// TIA Portal project "PROGETTO_TISC_FOSCHILLO_CUOMO" (V17)
// Vorlageprojekt für das Buch mit Zielsystem S7-1200

(* hardware
DEVICE "S7-1200-Station_1"  S7-1200 Station
   slot 0: "Baugruppenträger_0"  Rack  V1.0
   slot 1: "PLC_1"  CPU 1214C DC/DC/DC  6ES7 214-1AG40-0XB0  V4.5
DEVICE "HMI_1"  TP900 Comfort
   slot 0: "HMI_1"  TP900 Comfort  6AV2 124-0JC01-0AX0  17.0.0.0
   slot 1: "HMI_RT_1"  TP900 Comfort  6AV2 124-0JC01-0AX0  17.0.0.0
   slot 5: "HMI_1.IE_CP_1"  PROFINET Interface  17.0.0.0
      slot 1: "PROFINET Interface_1"  PROFINET Interface
         slot 1: "Port_1"  Port
         slot 2: "Port_2"  Port
   slot 7: "HMI_1.MPI/DP_CP_1"  MPI/DP Interface  17.0.0.0
*)

// ===== PLC "PLC_1"  CPU 1214C DC/DC/DC =====

VAR_GLOBAL   // PLC tag table "Standard-Variablentabelle"
   "Tag_1" AT %A0.0 : Bool;
   "Tag_2" AT %E0.0 : Bool;
   "Tag_3" AT %E0.1 : Bool;
   "PIANO_0" AT %I0.2 : Bool;
   "PIANO1_SLOW" AT %I0.3 : Bool;
   "PIANO1_STOP" AT %I0.4 : Bool;
   "PIANO2_SLOW" AT %I0.5 : Bool;
   "PIANO2_STOP" AT %I0.6 : Bool;
   "BASE_UP" AT %Q0.1 : Bool;
   "BASE_DOWN" AT %Q0.2 : Bool;
   "BASE_SLOW" AT %Q0.3 : Bool;
   "SENS_DX" AT %I0.7 : Bool;
   "SENS_SX" AT %I1.0 : Bool;
   "SPOSTA_DX" AT %Q0.4 : Bool;
   "SPOSTA_SX" AT %Q0.5 : Bool;
   "SPINGI_INIZIO" AT %I1.1 : Bool;
   "SPINGI_FINE" AT %I1.2 : Bool;
   "SENS_SPINGI" AT %I1.3 : Bool;
   "SPINGI" AT %Q0.6 : Bool;
   "PRONTO_CONS" AT %I1.4 : Bool;
   "AVA" AT %Q0.7 : Bool;
   "H1" AT %I1.5 : Bool;
   "H2" AT %I1.6 : Bool;
   "AVA1" AT %Q1.0 : Bool;
   "CONS_ELEV" AT %I1.7 : Bool;
   "RICEVUTO_P1" AT %I2.0 : Bool;
   "RICEVUTO_P2" AT %I2.1 : Bool;
   "AVA2" AT %Q1.1 : Bool;
   "AVA3" AT %Q1.2 : Bool;
   "Tag_4" AT %M1.0 : Bool;
   "Tag_5" AT %M1.1 : Bool;
   "pezzi_lavorati_NP1" AT %MW16 : Int;
   "pezzi_lavorati_NP2" AT %MW18 : Int;
END_VAR

DATA_BLOCK "MS0_DB"   // DB1
{ S7_Optimized_Access := 'TRUE' }
VERSION : 0.1
// stored: InstanceOfName MECCANISMO DI SPOSTAMENTO
"MECCANISMO DI SPOSTAMENTO"
BEGIN
END_DATA_BLOCK

DATA_BLOCK "P_DB"   // DB2
{ S7_Optimized_Access := 'TRUE' }
VERSION : 0.1
// stored: InstanceOfName Pusher
"Pusher"
BEGIN
END_DATA_BLOCK

DATA_BLOCK "BR0_DB"   // DB3
{ S7_Optimized_Access := 'TRUE' }
VERSION : 0.1
// stored: InstanceOfName Base con rulliera
"Base con rulliera"
BEGIN
END_DATA_BLOCK

DATA_BLOCK "N2_DB"   // DB4
{ S7_Optimized_Access := 'TRUE' }
VERSION : 0.1
// stored: InstanceOfName Nastro_2
"Nastro_2"
BEGIN
END_DATA_BLOCK

DATA_BLOCK "N1_DB"   // DB5
{ S7_Optimized_Access := 'TRUE' }
VERSION : 0.1
// stored: InstanceOfName Nastro_1
"Nastro_1"
BEGIN
END_DATA_BLOCK

DATA_BLOCK "NP1_DB"   // DB7
{ S7_Optimized_Access := 'TRUE' }
VERSION : 0.1
// stored: InstanceOfName nastri_sup
"nastri_sup"
BEGIN
END_DATA_BLOCK

DATA_BLOCK "NP2_DB"   // DB8
{ S7_Optimized_Access := 'TRUE' }
VERSION : 0.1
// stored: InstanceOfName nastri_sup
"nastri_sup"
BEGIN
END_DATA_BLOCK

DATA_BLOCK "nastri_sup_DB"   // DB9
{ S7_Optimized_Access := 'TRUE' }
VERSION : 0.1
// stored: InstanceOfName nastri_sup
"nastri_sup"
BEGIN
END_DATA_BLOCK

FUNCTION_BLOCK "MECCANISMO DI SPOSTAMENTO"   // FB1, LAD
{ S7_Optimized_Access := 'TRUE' }
VERSION : 0.1
   VAR_INPUT
      consegnato : Bool;
      ferma2 : Bool;
      ferma1 : Bool;
      PIANO_0 : Bool;
      PIANO1_SLOW : Bool;
      PIANO1_STOP : Bool;
      PIANO2_SLOW : Bool;
      sali_ok : Bool;
      PIANO2_STOP : Bool;
   END_VAR
   VAR_OUTPUT
      down_ok : Bool;
      BASE_UP : Bool;
      BASE_DOWN : Bool;
      pronto_ferma : Bool;
      BASE_SLOW : Bool;
   END_VAR
   VAR
      initVar : Bool;
      f0 : Bool;
      f1 : Bool;
      f2 : Bool;
      f3 : Bool;
      f4 : Bool;
      f5 : Bool;
      f6 : Bool;
      f7 : Bool;
      t1 : Bool;
      t2 : Bool;
      t3 : Bool;
      t4 : Bool;
      t5 : Bool;
      t6 : Bool;
      t7 : Bool;
      t8 : Bool;
      t9 : Bool;
   END_VAR
BEGIN

REGION Network 1: inizializzazione fase F0
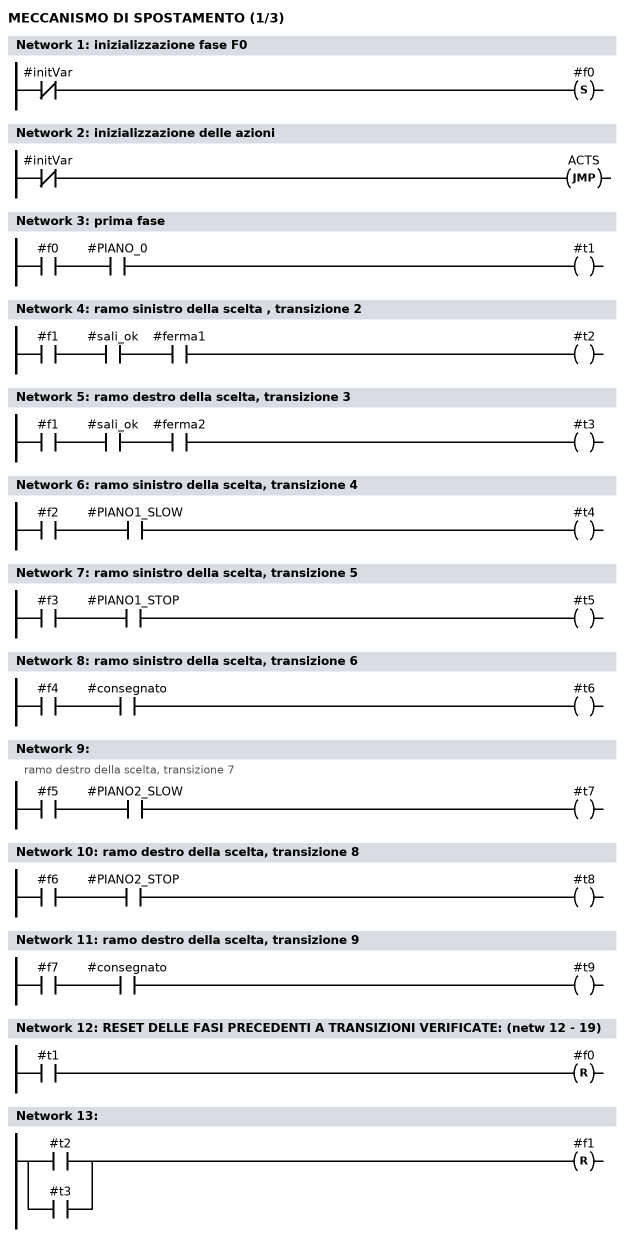
   RUNG wire#powerrail
      I_Contact( #initVar )
      S_Coil( #f0 )
   END_RUNG
   // the same network as SCL:
   IF NOT #initVar THEN #f0 := TRUE; END_IF;
END_REGION

REGION Network 2: inizializzazione delle azioni
   RUNG wire#powerrail
      I_Contact( #initVar )
      JumpCoil( ACTS )
   END_RUNG
   // the same network as SCL:
   IF NOT #initVar THEN GOTO ACTS; END_IF;
END_REGION

REGION Network 3: prima fase
   RUNG wire#powerrail
      Contact( #f0 )
      Contact( #PIANO_0 )
      Coil( #t1 )
   END_RUNG
   // the same network as SCL:
   #t1 := #f0 AND #PIANO_0;
END_REGION

REGION Network 4: ramo sinistro della scelta , transizione 2
   RUNG wire#powerrail
      Contact( #f1 )
      Contact( #sali_ok )
      Contact( #ferma1 )
      Coil( #t2 )
   END_RUNG
   // the same network as SCL:
   #t2 := #f1 AND #sali_ok AND #ferma1;
END_REGION

REGION Network 5: ramo destro della scelta, transizione 3
   RUNG wire#powerrail
      Contact( #f1 )
      Contact( #sali_ok )
      Contact( #ferma2 )
      Coil( #t3 )
   END_RUNG
   // the same network as SCL:
   #t3 := #f1 AND #sali_ok AND #ferma2;
END_REGION

REGION Network 6: ramo sinistro della scelta, transizione 4
   RUNG wire#powerrail
      Contact( #f2 )
      Contact( #PIANO1_SLOW )
      Coil( #t4 )
   END_RUNG
   // the same network as SCL:
   #t4 := #f2 AND #PIANO1_SLOW;
END_REGION

REGION Network 7: ramo sinistro della scelta, transizione 5
   RUNG wire#powerrail
      Contact( #f3 )
      Contact( #PIANO1_STOP )
      Coil( #t5 )
   END_RUNG
   // the same network as SCL:
   #t5 := #f3 AND #PIANO1_STOP;
END_REGION

REGION Network 8: ramo sinistro della scelta, transizione 6
   RUNG wire#powerrail
      Contact( #f4 )
      Contact( #consegnato )
      Coil( #t6 )
   END_RUNG
   // the same network as SCL:
   #t6 := #f4 AND #consegnato;
END_REGION

REGION Network 9
   // ramo destro della scelta, transizione 7
   RUNG wire#powerrail
      Contact( #f5 )
      Contact( #PIANO2_SLOW )
      Coil( #t7 )
   END_RUNG
   // the same network as SCL:
   #t7 := #f5 AND #PIANO2_SLOW;
END_REGION

REGION Network 10: ramo destro della scelta, transizione 8
   RUNG wire#powerrail
      Contact( #f6 )
      Contact( #PIANO2_STOP )
      Coil( #t8 )
   END_RUNG
   // the same network as SCL:
   #t8 := #f6 AND #PIANO2_STOP;
END_REGION

REGION Network 11: ramo destro della scelta, transizione 9
   RUNG wire#powerrail
      Contact( #f7 )
      Contact( #consegnato )
      Coil( #t9 )
   END_RUNG
   // the same network as SCL:
   #t9 := #f7 AND #consegnato;
END_REGION

REGION Network 12: RESET DELLE FASI PRECEDENTI A TRANSIZIONI VERIFICATE: (netw 12 - 19)
   RUNG wire#powerrail
      Contact( #t1 )
      R_Coil( #f0 )
   END_RUNG
   // the same network as SCL:
   IF #t1 THEN #f0 := FALSE; END_IF;
END_REGION

REGION Network 13
   RUNG wire#powerrail
      Contact( #t2 )
      wire#w1
      R_Coil( #f1 )
   END_RUNG
   RUNG wire#powerrail
      Contact( #t3 )
   END_RUNG wire#w1
   // the same network as SCL:
   IF #t2 OR #t3 THEN #f1 := FALSE; END_IF;
END_REGION

REGION Network 14
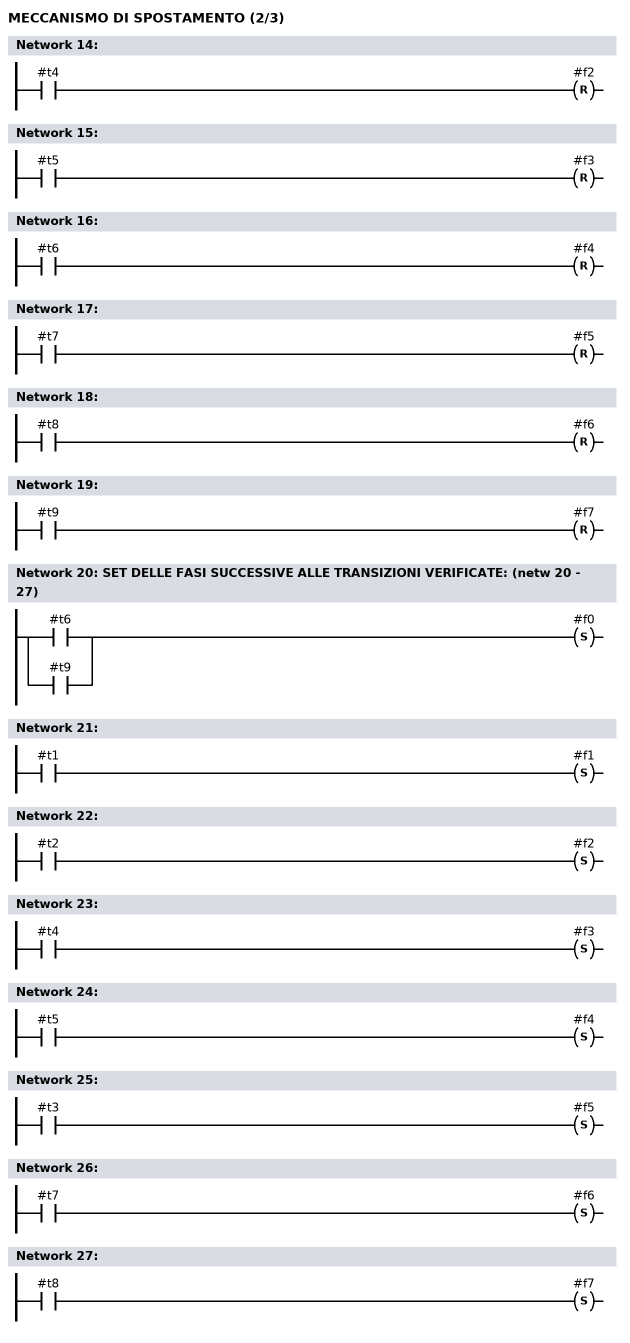
   RUNG wire#powerrail
      Contact( #t4 )
      R_Coil( #f2 )
   END_RUNG
   // the same network as SCL:
   IF #t4 THEN #f2 := FALSE; END_IF;
END_REGION

REGION Network 15
   RUNG wire#powerrail
      Contact( #t5 )
      R_Coil( #f3 )
   END_RUNG
   // the same network as SCL:
   IF #t5 THEN #f3 := FALSE; END_IF;
END_REGION

REGION Network 16
   RUNG wire#powerrail
      Contact( #t6 )
      R_Coil( #f4 )
   END_RUNG
   // the same network as SCL:
   IF #t6 THEN #f4 := FALSE; END_IF;
END_REGION

REGION Network 17
   RUNG wire#powerrail
      Contact( #t7 )
      R_Coil( #f5 )
   END_RUNG
   // the same network as SCL:
   IF #t7 THEN #f5 := FALSE; END_IF;
END_REGION

REGION Network 18
   RUNG wire#powerrail
      Contact( #t8 )
      R_Coil( #f6 )
   END_RUNG
   // the same network as SCL:
   IF #t8 THEN #f6 := FALSE; END_IF;
END_REGION

REGION Network 19
   RUNG wire#powerrail
      Contact( #t9 )
      R_Coil( #f7 )
   END_RUNG
   // the same network as SCL:
   IF #t9 THEN #f7 := FALSE; END_IF;
END_REGION

REGION Network 20: SET DELLE FASI SUCCESSIVE ALLE TRANSIZIONI VERIFICATE: (netw 20 - 27)
   RUNG wire#powerrail
      Contact( #t6 )
      wire#w1
      S_Coil( #f0 )
   END_RUNG
   RUNG wire#powerrail
      Contact( #t9 )
   END_RUNG wire#w1
   // the same network as SCL:
   IF #t6 OR #t9 THEN #f0 := TRUE; END_IF;
END_REGION

REGION Network 21
   RUNG wire#powerrail
      Contact( #t1 )
      S_Coil( #f1 )
   END_RUNG
   // the same network as SCL:
   IF #t1 THEN #f1 := TRUE; END_IF;
END_REGION

REGION Network 22
   RUNG wire#powerrail
      Contact( #t2 )
      S_Coil( #f2 )
   END_RUNG
   // the same network as SCL:
   IF #t2 THEN #f2 := TRUE; END_IF;
END_REGION

REGION Network 23
   RUNG wire#powerrail
      Contact( #t4 )
      S_Coil( #f3 )
   END_RUNG
   // the same network as SCL:
   IF #t4 THEN #f3 := TRUE; END_IF;
END_REGION

REGION Network 24
   RUNG wire#powerrail
      Contact( #t5 )
      S_Coil( #f4 )
   END_RUNG
   // the same network as SCL:
   IF #t5 THEN #f4 := TRUE; END_IF;
END_REGION

REGION Network 25
   RUNG wire#powerrail
      Contact( #t3 )
      S_Coil( #f5 )
   END_RUNG
   // the same network as SCL:
   IF #t3 THEN #f5 := TRUE; END_IF;
END_REGION

REGION Network 26
   RUNG wire#powerrail
      Contact( #t7 )
      S_Coil( #f6 )
   END_RUNG
   // the same network as SCL:
   IF #t7 THEN #f6 := TRUE; END_IF;
END_REGION

REGION Network 27
   RUNG wire#powerrail
      Contact( #t8 )
      S_Coil( #f7 )
   END_RUNG
   // the same network as SCL:
   IF #t8 THEN #f7 := TRUE; END_IF;
END_REGION

REGION Network 28: INIZIALIZZAZIONE DELLE AZIONI CORRISPONDENTI AD OGNI FASE:
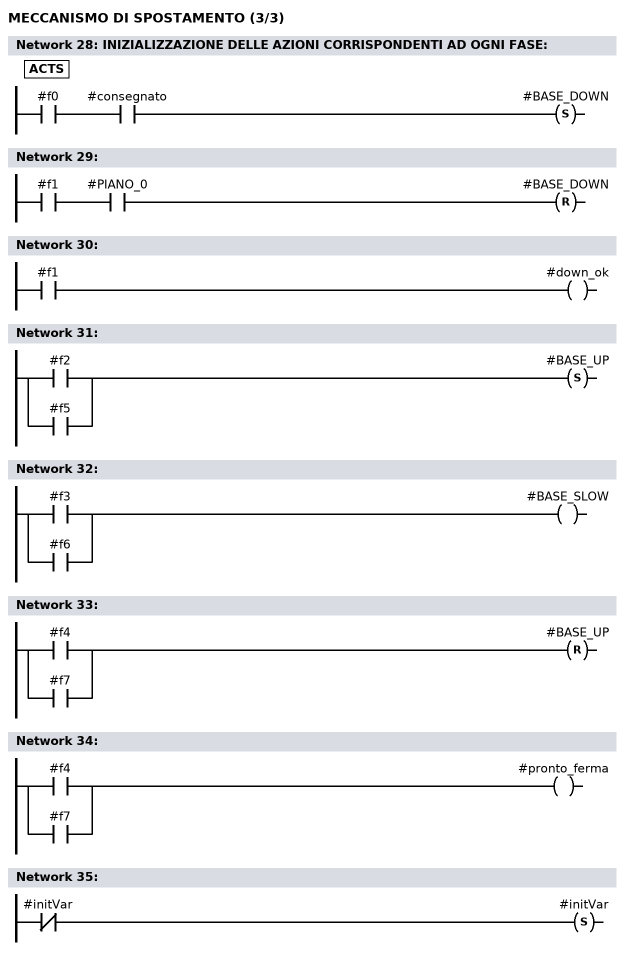
   Label( ACTS )
   RUNG wire#powerrail
      Contact( #f0 )
      Contact( #consegnato )
      S_Coil( #BASE_DOWN )
   END_RUNG
   // the same network as SCL:
   ACTS:
   IF #f0 AND #consegnato THEN #BASE_DOWN := TRUE; END_IF;
END_REGION

REGION Network 29
   RUNG wire#powerrail
      Contact( #f1 )
      Contact( #PIANO_0 )
      R_Coil( #BASE_DOWN )
   END_RUNG
   // the same network as SCL:
   IF #f1 AND #PIANO_0 THEN #BASE_DOWN := FALSE; END_IF;
END_REGION

REGION Network 30
   RUNG wire#powerrail
      Contact( #f1 )
      Coil( #down_ok )
   END_RUNG
   // the same network as SCL:
   #down_ok := #f1;
END_REGION

REGION Network 31
   RUNG wire#powerrail
      Contact( #f2 )
      wire#w1
      S_Coil( #BASE_UP )
   END_RUNG
   RUNG wire#powerrail
      Contact( #f5 )
   END_RUNG wire#w1
   // the same network as SCL:
   IF #f2 OR #f5 THEN #BASE_UP := TRUE; END_IF;
END_REGION

REGION Network 32
   RUNG wire#powerrail
      Contact( #f3 )
      wire#w1
      Coil( #BASE_SLOW )
   END_RUNG
   RUNG wire#powerrail
      Contact( #f6 )
   END_RUNG wire#w1
   // the same network as SCL:
   #BASE_SLOW := #f3 OR #f6;
END_REGION

REGION Network 33
   RUNG wire#powerrail
      Contact( #f4 )
      wire#w1
      R_Coil( #BASE_UP )
   END_RUNG
   RUNG wire#powerrail
      Contact( #f7 )
   END_RUNG wire#w1
   // the same network as SCL:
   IF #f4 OR #f7 THEN #BASE_UP := FALSE; END_IF;
END_REGION

REGION Network 34
   RUNG wire#powerrail
      Contact( #f4 )
      wire#w1
      Coil( #pronto_ferma )
   END_RUNG
   RUNG wire#powerrail
      Contact( #f7 )
   END_RUNG wire#w1
   // the same network as SCL:
   #pronto_ferma := #f4 OR #f7;
END_REGION

REGION Network 35
   RUNG wire#powerrail
      I_Contact( #initVar )
      S_Coil( #initVar )
   END_RUNG
   // the same network as SCL:
   IF NOT #initVar THEN #initVar := TRUE; END_IF;
END_REGION
END_FUNCTION_BLOCK

FUNCTION_BLOCK "Base con rulliera"   // FB2, LAD
{ S7_Optimized_Access := 'TRUE' }
VERSION : 0.1
   VAR_INPUT
      SENS_SX : Bool;
      SENS_DX : Bool;
      OK_PRENDI : Bool;
      OK_RILASCIA : Bool;
      FINITO1 : Bool;
      FINITO2 : Bool;
   END_VAR
   VAR_OUTPUT
      SPOSTA_DX : Bool;
      SPOSTA_SX : Bool;
      FINE_PRENDI : Bool;
      FINE_CONSEGNA : Bool;
   END_VAR
   VAR
      InitVar : Bool;
      f0 : Bool;
      f1 : Bool;
      f2 : Bool;
      f3 : Bool;
      f4 : Bool;
      t0 : Bool;
      t1 : Bool;
      t2 : Bool;
      t3 : Bool;
      t4 : Bool;
      t5 : Bool;
      SENS_SX_FTRIG : F_TRIG;
   END_VAR
BEGIN

REGION Network 1: INIZIALIZZAZIONE FASE INIZIALE
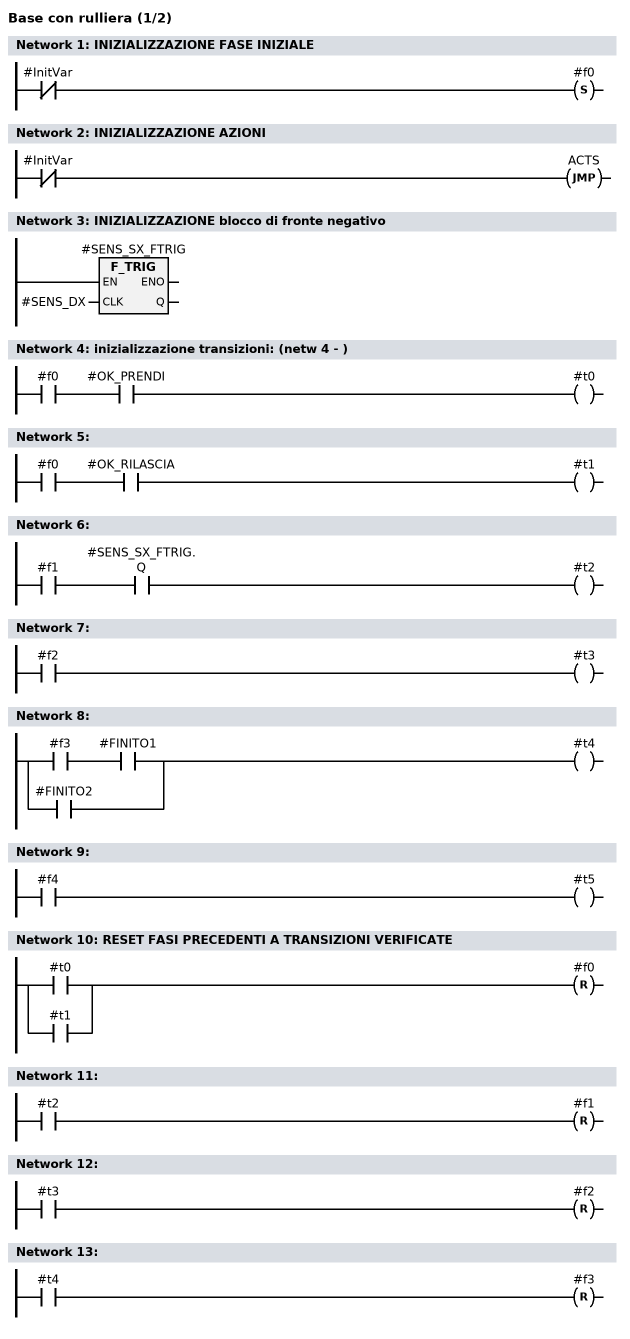
   RUNG wire#powerrail
      I_Contact( #InitVar )
      S_Coil( #f0 )
   END_RUNG
   // the same network as SCL:
   IF NOT #InitVar THEN #f0 := TRUE; END_IF;
END_REGION

REGION Network 2: INIZIALIZZAZIONE AZIONI
   RUNG wire#powerrail
      I_Contact( #InitVar )
      JumpCoil( ACTS )
   END_RUNG
   // the same network as SCL:
   IF NOT #InitVar THEN GOTO ACTS; END_IF;
END_REGION

REGION Network 3: INIZIALIZZAZIONE blocco di fronte negativo
   #SENS_SX_FTRIG(CLK := #SENS_DX);   // F_TRIG
END_REGION

REGION Network 4: inizializzazione transizioni: (netw 4 - )
   RUNG wire#powerrail
      Contact( #f0 )
      Contact( #OK_PRENDI )
      Coil( #t0 )
   END_RUNG
   // the same network as SCL:
   #t0 := #f0 AND #OK_PRENDI;
END_REGION

REGION Network 5
   RUNG wire#powerrail
      Contact( #f0 )
      Contact( #OK_RILASCIA )
      Coil( #t1 )
   END_RUNG
   // the same network as SCL:
   #t1 := #f0 AND #OK_RILASCIA;
END_REGION

REGION Network 6
   RUNG wire#powerrail
      Contact( #f1 )
      Contact( #SENS_SX_FTRIG.Q )
      Coil( #t2 )
   END_RUNG
   // the same network as SCL:
   #t2 := #f1 AND #SENS_SX_FTRIG.Q;
END_REGION

REGION Network 7
   RUNG wire#powerrail
      Contact( #f2 )
      Coil( #t3 )
   END_RUNG
   // the same network as SCL:
   #t3 := #f2;
END_REGION

REGION Network 8
   RUNG wire#powerrail
      Contact( #f3 )
      Contact( #FINITO1 )
      wire#w1
      Coil( #t4 )
   END_RUNG
   RUNG wire#powerrail
      Contact( #FINITO2 )
   END_RUNG wire#w1
   // the same network as SCL:
   #t4 := (#f3 AND #FINITO1) OR #FINITO2;
END_REGION

REGION Network 9
   RUNG wire#powerrail
      Contact( #f4 )
      Coil( #t5 )
   END_RUNG
   // the same network as SCL:
   #t5 := #f4;
END_REGION

REGION Network 10: RESET FASI PRECEDENTI A TRANSIZIONI VERIFICATE
   RUNG wire#powerrail
      Contact( #t0 )
      wire#w1
      R_Coil( #f0 )
   END_RUNG
   RUNG wire#powerrail
      Contact( #t1 )
   END_RUNG wire#w1
   // the same network as SCL:
   IF #t0 OR #t1 THEN #f0 := FALSE; END_IF;
END_REGION

REGION Network 11
   RUNG wire#powerrail
      Contact( #t2 )
      R_Coil( #f1 )
   END_RUNG
   // the same network as SCL:
   IF #t2 THEN #f1 := FALSE; END_IF;
END_REGION

REGION Network 12
   RUNG wire#powerrail
      Contact( #t3 )
      R_Coil( #f2 )
   END_RUNG
   // the same network as SCL:
   IF #t3 THEN #f2 := FALSE; END_IF;
END_REGION

REGION Network 13
   RUNG wire#powerrail
      Contact( #t4 )
      R_Coil( #f3 )
   END_RUNG
   // the same network as SCL:
   IF #t4 THEN #f3 := FALSE; END_IF;
END_REGION

REGION Network 14
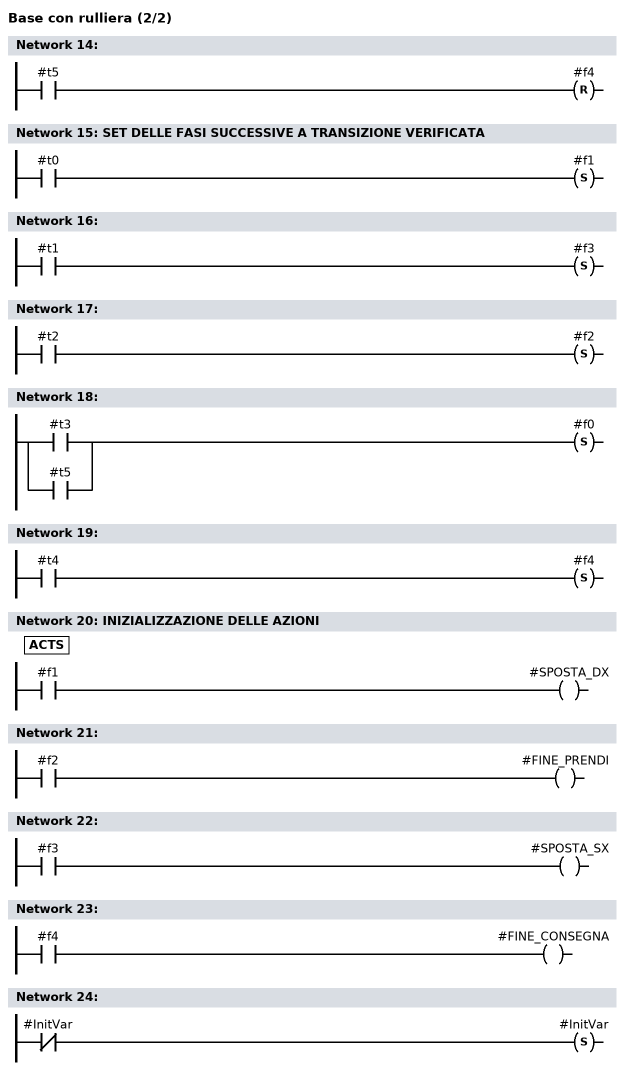
   RUNG wire#powerrail
      Contact( #t5 )
      R_Coil( #f4 )
   END_RUNG
   // the same network as SCL:
   IF #t5 THEN #f4 := FALSE; END_IF;
END_REGION

REGION Network 15: SET DELLE FASI SUCCESSIVE A TRANSIZIONE VERIFICATA
   RUNG wire#powerrail
      Contact( #t0 )
      S_Coil( #f1 )
   END_RUNG
   // the same network as SCL:
   IF #t0 THEN #f1 := TRUE; END_IF;
END_REGION

REGION Network 16
   RUNG wire#powerrail
      Contact( #t1 )
      S_Coil( #f3 )
   END_RUNG
   // the same network as SCL:
   IF #t1 THEN #f3 := TRUE; END_IF;
END_REGION

REGION Network 17
   RUNG wire#powerrail
      Contact( #t2 )
      S_Coil( #f2 )
   END_RUNG
   // the same network as SCL:
   IF #t2 THEN #f2 := TRUE; END_IF;
END_REGION

REGION Network 18
   RUNG wire#powerrail
      Contact( #t3 )
      wire#w1
      S_Coil( #f0 )
   END_RUNG
   RUNG wire#powerrail
      Contact( #t5 )
   END_RUNG wire#w1
   // the same network as SCL:
   IF #t3 OR #t5 THEN #f0 := TRUE; END_IF;
END_REGION

REGION Network 19
   RUNG wire#powerrail
      Contact( #t4 )
      S_Coil( #f4 )
   END_RUNG
   // the same network as SCL:
   IF #t4 THEN #f4 := TRUE; END_IF;
END_REGION

REGION Network 20: INIZIALIZZAZIONE DELLE AZIONI
   Label( ACTS )
   RUNG wire#powerrail
      Contact( #f1 )
      Coil( #SPOSTA_DX )
   END_RUNG
   // the same network as SCL:
   ACTS:
   #SPOSTA_DX := #f1;
END_REGION

REGION Network 21
   RUNG wire#powerrail
      Contact( #f2 )
      Coil( #FINE_PRENDI )
   END_RUNG
   // the same network as SCL:
   #FINE_PRENDI := #f2;
END_REGION

REGION Network 22
   RUNG wire#powerrail
      Contact( #f3 )
      Coil( #SPOSTA_SX )
   END_RUNG
   // the same network as SCL:
   #SPOSTA_SX := #f3;
END_REGION

REGION Network 23
   RUNG wire#powerrail
      Contact( #f4 )
      Coil( #FINE_CONSEGNA )
   END_RUNG
   // the same network as SCL:
   #FINE_CONSEGNA := #f4;
END_REGION

REGION Network 24
   RUNG wire#powerrail
      I_Contact( #InitVar )
      S_Coil( #InitVar )
   END_RUNG
   // the same network as SCL:
   IF NOT #InitVar THEN #InitVar := TRUE; END_IF;
END_REGION
END_FUNCTION_BLOCK

FUNCTION_BLOCK "Nastro_2"   // FB3, LAD
{ S7_Optimized_Access := 'TRUE' }
VERSION : 0.1
   VAR_INPUT
      pacco_cons : Bool;
      h1 : Bool;
      h2 : Bool;
      consegna_elevatore : Bool;
      consegna_ok : Bool;
      preso_ok : Bool;
   END_VAR
   VAR_OUTPUT
      ava : Bool;
      p_ricevere : Bool;
      ferma_1 : Bool;
      ferma_2 : Bool;
   END_VAR
   VAR
      iniz : Bool;
      f1 : Bool;
      t1 : Bool;
      t2 : Bool;
      f2 : Bool;
      t3 : Bool;
      f5 : Bool;
      t4 : Bool;
      f3 : Bool;
      t5 : Bool;
      f6 : Bool;
      t6 : Bool;
      f4 : Bool;
      t7 : Bool;
      f7 : Bool;
      t8 : Bool;
      f8 : Bool;
      f9 : Bool;
      t9 : Bool;
      t10 : Bool;
   END_VAR
BEGIN

REGION Network 1
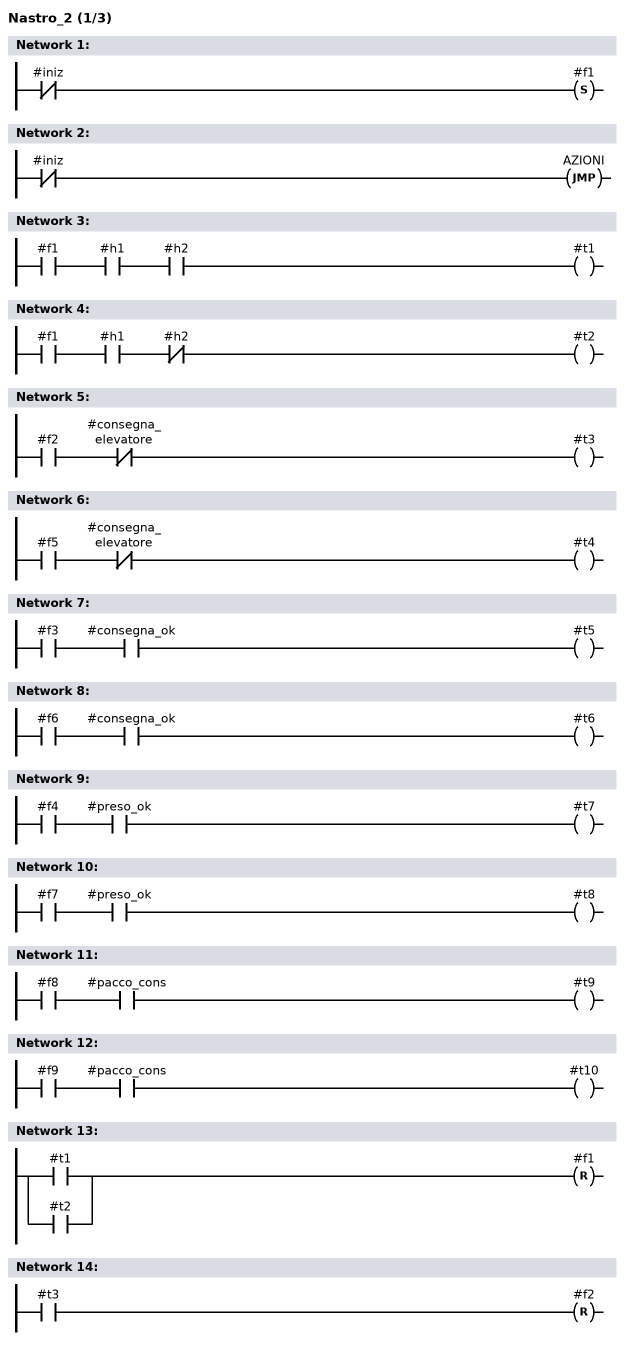
   RUNG wire#powerrail
      I_Contact( #iniz )
      S_Coil( #f1 )
   END_RUNG
   // the same network as SCL:
   IF NOT #iniz THEN #f1 := TRUE; END_IF;
END_REGION

REGION Network 2
   RUNG wire#powerrail
      I_Contact( #iniz )
      JumpCoil( AZIONI )
   END_RUNG
   // the same network as SCL:
   IF NOT #iniz THEN GOTO AZIONI; END_IF;
END_REGION

REGION Network 3
   RUNG wire#powerrail
      Contact( #f1 )
      Contact( #h1 )
      Contact( #h2 )
      Coil( #t1 )
   END_RUNG
   // the same network as SCL:
   #t1 := #f1 AND #h1 AND #h2;
END_REGION

REGION Network 4
   RUNG wire#powerrail
      Contact( #f1 )
      Contact( #h1 )
      I_Contact( #h2 )
      Coil( #t2 )
   END_RUNG
   // the same network as SCL:
   #t2 := #f1 AND #h1 AND NOT #h2;
END_REGION

REGION Network 5
   RUNG wire#powerrail
      Contact( #f2 )
      I_Contact( #consegna_elevatore )
      Coil( #t3 )
   END_RUNG
   // the same network as SCL:
   #t3 := #f2 AND NOT #consegna_elevatore;
END_REGION

REGION Network 6
   RUNG wire#powerrail
      Contact( #f5 )
      I_Contact( #consegna_elevatore )
      Coil( #t4 )
   END_RUNG
   // the same network as SCL:
   #t4 := #f5 AND NOT #consegna_elevatore;
END_REGION

REGION Network 7
   RUNG wire#powerrail
      Contact( #f3 )
      Contact( #consegna_ok )
      Coil( #t5 )
   END_RUNG
   // the same network as SCL:
   #t5 := #f3 AND #consegna_ok;
END_REGION

REGION Network 8
   RUNG wire#powerrail
      Contact( #f6 )
      Contact( #consegna_ok )
      Coil( #t6 )
   END_RUNG
   // the same network as SCL:
   #t6 := #f6 AND #consegna_ok;
END_REGION

REGION Network 9
   RUNG wire#powerrail
      Contact( #f4 )
      Contact( #preso_ok )
      Coil( #t7 )
   END_RUNG
   // the same network as SCL:
   #t7 := #f4 AND #preso_ok;
END_REGION

REGION Network 10
   RUNG wire#powerrail
      Contact( #f7 )
      Contact( #preso_ok )
      Coil( #t8 )
   END_RUNG
   // the same network as SCL:
   #t8 := #f7 AND #preso_ok;
END_REGION

REGION Network 11
   RUNG wire#powerrail
      Contact( #f8 )
      Contact( #pacco_cons )
      Coil( #t9 )
   END_RUNG
   // the same network as SCL:
   #t9 := #f8 AND #pacco_cons;
END_REGION

REGION Network 12
   RUNG wire#powerrail
      Contact( #f9 )
      Contact( #pacco_cons )
      Coil( #t10 )
   END_RUNG
   // the same network as SCL:
   #t10 := #f9 AND #pacco_cons;
END_REGION

REGION Network 13
   RUNG wire#powerrail
      Contact( #t1 )
      wire#w1
      R_Coil( #f1 )
   END_RUNG
   RUNG wire#powerrail
      Contact( #t2 )
   END_RUNG wire#w1
   // the same network as SCL:
   IF #t1 OR #t2 THEN #f1 := FALSE; END_IF;
END_REGION

REGION Network 14
   RUNG wire#powerrail
      Contact( #t3 )
      R_Coil( #f2 )
   END_RUNG
   // the same network as SCL:
   IF #t3 THEN #f2 := FALSE; END_IF;
END_REGION

REGION Network 15
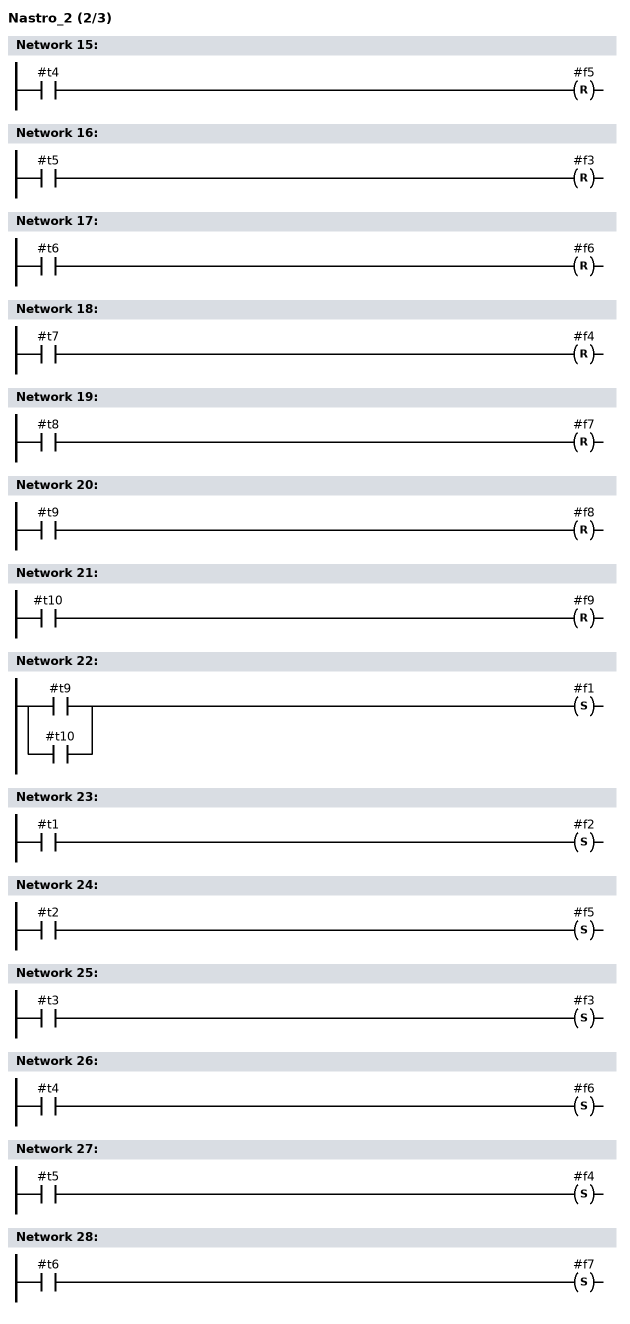
   RUNG wire#powerrail
      Contact( #t4 )
      R_Coil( #f5 )
   END_RUNG
   // the same network as SCL:
   IF #t4 THEN #f5 := FALSE; END_IF;
END_REGION

REGION Network 16
   RUNG wire#powerrail
      Contact( #t5 )
      R_Coil( #f3 )
   END_RUNG
   // the same network as SCL:
   IF #t5 THEN #f3 := FALSE; END_IF;
END_REGION

REGION Network 17
   RUNG wire#powerrail
      Contact( #t6 )
      R_Coil( #f6 )
   END_RUNG
   // the same network as SCL:
   IF #t6 THEN #f6 := FALSE; END_IF;
END_REGION

REGION Network 18
   RUNG wire#powerrail
      Contact( #t7 )
      R_Coil( #f4 )
   END_RUNG
   // the same network as SCL:
   IF #t7 THEN #f4 := FALSE; END_IF;
END_REGION

REGION Network 19
   RUNG wire#powerrail
      Contact( #t8 )
      R_Coil( #f7 )
   END_RUNG
   // the same network as SCL:
   IF #t8 THEN #f7 := FALSE; END_IF;
END_REGION

REGION Network 20
   RUNG wire#powerrail
      Contact( #t9 )
      R_Coil( #f8 )
   END_RUNG
   // the same network as SCL:
   IF #t9 THEN #f8 := FALSE; END_IF;
END_REGION

REGION Network 21
   RUNG wire#powerrail
      Contact( #t10 )
      R_Coil( #f9 )
   END_RUNG
   // the same network as SCL:
   IF #t10 THEN #f9 := FALSE; END_IF;
END_REGION

REGION Network 22
   RUNG wire#powerrail
      Contact( #t9 )
      wire#w1
      S_Coil( #f1 )
   END_RUNG
   RUNG wire#powerrail
      Contact( #t10 )
   END_RUNG wire#w1
   // the same network as SCL:
   IF #t9 OR #t10 THEN #f1 := TRUE; END_IF;
END_REGION

REGION Network 23
   RUNG wire#powerrail
      Contact( #t1 )
      S_Coil( #f2 )
   END_RUNG
   // the same network as SCL:
   IF #t1 THEN #f2 := TRUE; END_IF;
END_REGION

REGION Network 24
   RUNG wire#powerrail
      Contact( #t2 )
      S_Coil( #f5 )
   END_RUNG
   // the same network as SCL:
   IF #t2 THEN #f5 := TRUE; END_IF;
END_REGION

REGION Network 25
   RUNG wire#powerrail
      Contact( #t3 )
      S_Coil( #f3 )
   END_RUNG
   // the same network as SCL:
   IF #t3 THEN #f3 := TRUE; END_IF;
END_REGION

REGION Network 26
   RUNG wire#powerrail
      Contact( #t4 )
      S_Coil( #f6 )
   END_RUNG
   // the same network as SCL:
   IF #t4 THEN #f6 := TRUE; END_IF;
END_REGION

REGION Network 27
   RUNG wire#powerrail
      Contact( #t5 )
      S_Coil( #f4 )
   END_RUNG
   // the same network as SCL:
   IF #t5 THEN #f4 := TRUE; END_IF;
END_REGION

REGION Network 28
   RUNG wire#powerrail
      Contact( #t6 )
      S_Coil( #f7 )
   END_RUNG
   // the same network as SCL:
   IF #t6 THEN #f7 := TRUE; END_IF;
END_REGION

REGION Network 29
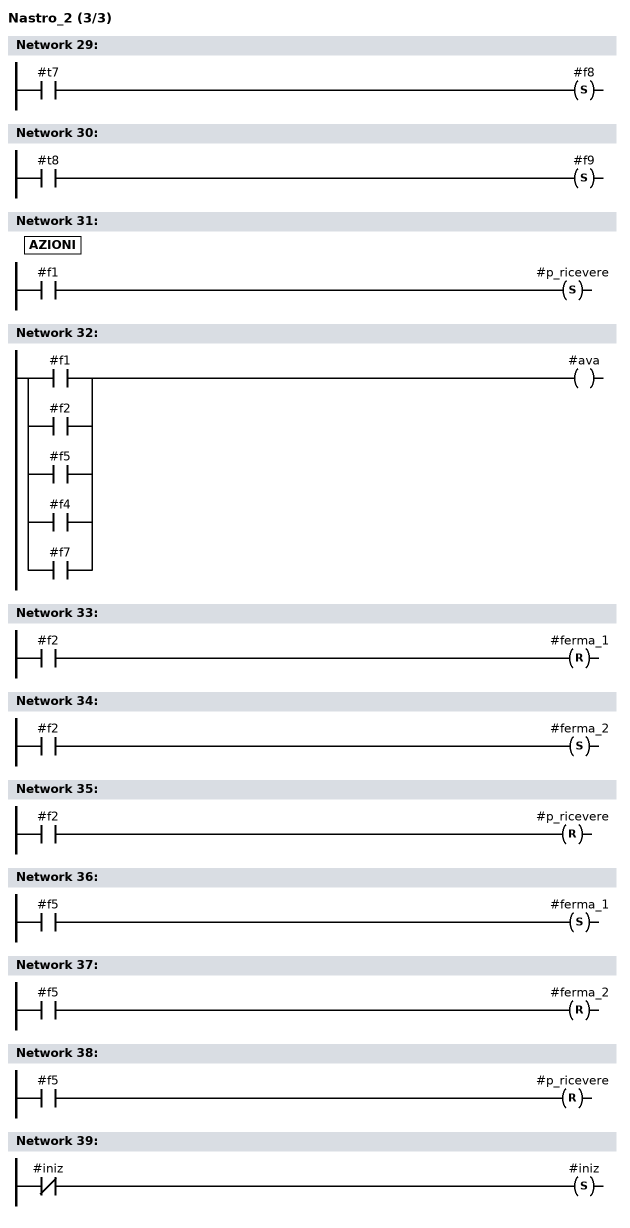
   RUNG wire#powerrail
      Contact( #t7 )
      S_Coil( #f8 )
   END_RUNG
   // the same network as SCL:
   IF #t7 THEN #f8 := TRUE; END_IF;
END_REGION

REGION Network 30
   RUNG wire#powerrail
      Contact( #t8 )
      S_Coil( #f9 )
   END_RUNG
   // the same network as SCL:
   IF #t8 THEN #f9 := TRUE; END_IF;
END_REGION

REGION Network 31
   Label( AZIONI )
   RUNG wire#powerrail
      Contact( #f1 )
      S_Coil( #p_ricevere )
   END_RUNG
   // the same network as SCL:
   AZIONI:
   IF #f1 THEN #p_ricevere := TRUE; END_IF;
END_REGION

REGION Network 32
   RUNG wire#powerrail
      Contact( #f1 )
      wire#w1
      Coil( #ava )
   END_RUNG
   RUNG wire#powerrail
      Contact( #f2 )
   END_RUNG wire#w1
   RUNG wire#powerrail
      Contact( #f5 )
   END_RUNG wire#w1
   RUNG wire#powerrail
      Contact( #f4 )
   END_RUNG wire#w1
   RUNG wire#powerrail
      Contact( #f7 )
   END_RUNG wire#w1
   // the same network as SCL:
   #ava := #f1 OR #f2 OR #f5 OR #f4 OR #f7;
END_REGION

REGION Network 33
   RUNG wire#powerrail
      Contact( #f2 )
      R_Coil( #ferma_1 )
   END_RUNG
   // the same network as SCL:
   IF #f2 THEN #ferma_1 := FALSE; END_IF;
END_REGION

REGION Network 34
   RUNG wire#powerrail
      Contact( #f2 )
      S_Coil( #ferma_2 )
   END_RUNG
   // the same network as SCL:
   IF #f2 THEN #ferma_2 := TRUE; END_IF;
END_REGION

REGION Network 35
   RUNG wire#powerrail
      Contact( #f2 )
      R_Coil( #p_ricevere )
   END_RUNG
   // the same network as SCL:
   IF #f2 THEN #p_ricevere := FALSE; END_IF;
END_REGION

REGION Network 36
   RUNG wire#powerrail
      Contact( #f5 )
      S_Coil( #ferma_1 )
   END_RUNG
   // the same network as SCL:
   IF #f5 THEN #ferma_1 := TRUE; END_IF;
END_REGION

REGION Network 37
   RUNG wire#powerrail
      Contact( #f5 )
      R_Coil( #ferma_2 )
   END_RUNG
   // the same network as SCL:
   IF #f5 THEN #ferma_2 := FALSE; END_IF;
END_REGION

REGION Network 38
   RUNG wire#powerrail
      Contact( #f5 )
      R_Coil( #p_ricevere )
   END_RUNG
   // the same network as SCL:
   IF #f5 THEN #p_ricevere := FALSE; END_IF;
END_REGION

REGION Network 39
   RUNG wire#powerrail
      I_Contact( #iniz )
      S_Coil( #iniz )
   END_RUNG
   // the same network as SCL:
   IF NOT #iniz THEN #iniz := TRUE; END_IF;
END_REGION
END_FUNCTION_BLOCK

FUNCTION_BLOCK "nastri_sup"   // FB4, LAD
{ S7_Optimized_Access := 'TRUE' }
VERSION : 0.1
   VAR_INPUT
      ricevuto_p : Bool;
   END_VAR
   VAR_OUTPUT
      ava : Bool;
      ricevuto_ok : Bool;
   END_VAR
   VAR
      iniz : Bool;
      f1 : Bool;
      ricevuto_RTRIG : R_TRIG;
      t1 : Bool;
      f2 : Bool;
      t2 : Bool;
   END_VAR
BEGIN

REGION Network 1
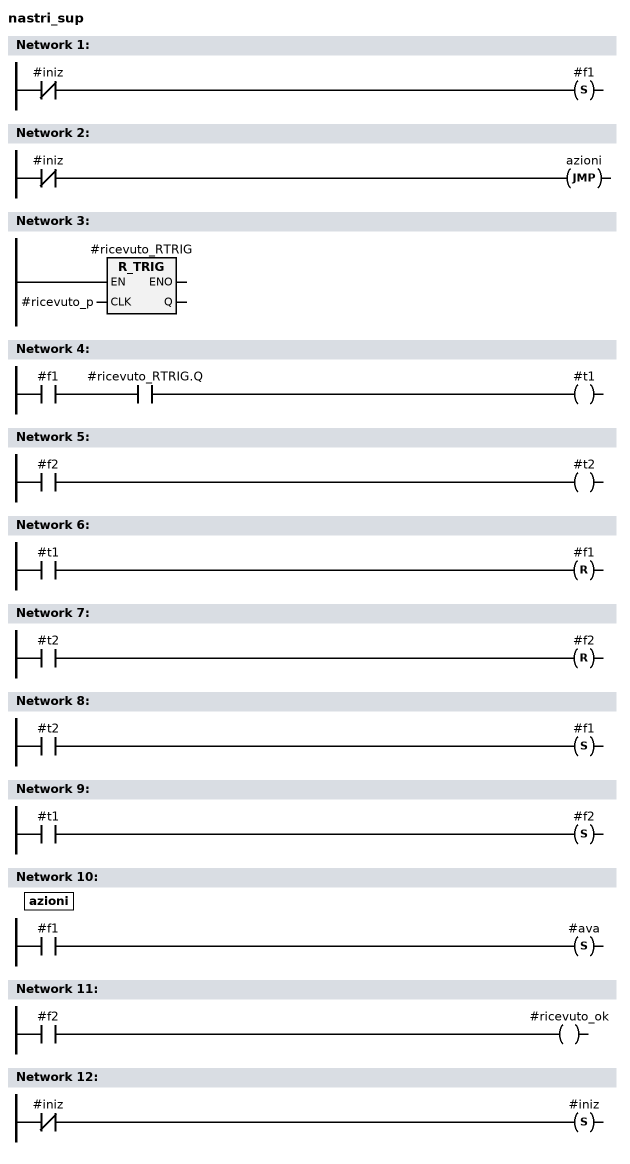
   RUNG wire#powerrail
      I_Contact( #iniz )
      S_Coil( #f1 )
   END_RUNG
   // the same network as SCL:
   IF NOT #iniz THEN #f1 := TRUE; END_IF;
END_REGION

REGION Network 2
   RUNG wire#powerrail
      I_Contact( #iniz )
      JumpCoil( azioni )
   END_RUNG
   // the same network as SCL:
   IF NOT #iniz THEN GOTO azioni; END_IF;
END_REGION

REGION Network 3
   #ricevuto_RTRIG(CLK := #ricevuto_p);   // R_TRIG
END_REGION

REGION Network 4
   RUNG wire#powerrail
      Contact( #f1 )
      Contact( #ricevuto_RTRIG.Q )
      Coil( #t1 )
   END_RUNG
   // the same network as SCL:
   #t1 := #f1 AND #ricevuto_RTRIG.Q;
END_REGION

REGION Network 5
   RUNG wire#powerrail
      Contact( #f2 )
      Coil( #t2 )
   END_RUNG
   // the same network as SCL:
   #t2 := #f2;
END_REGION

REGION Network 6
   RUNG wire#powerrail
      Contact( #t1 )
      R_Coil( #f1 )
   END_RUNG
   // the same network as SCL:
   IF #t1 THEN #f1 := FALSE; END_IF;
END_REGION

REGION Network 7
   RUNG wire#powerrail
      Contact( #t2 )
      R_Coil( #f2 )
   END_RUNG
   // the same network as SCL:
   IF #t2 THEN #f2 := FALSE; END_IF;
END_REGION

REGION Network 8
   RUNG wire#powerrail
      Contact( #t2 )
      S_Coil( #f1 )
   END_RUNG
   // the same network as SCL:
   IF #t2 THEN #f1 := TRUE; END_IF;
END_REGION

REGION Network 9
   RUNG wire#powerrail
      Contact( #t1 )
      S_Coil( #f2 )
   END_RUNG
   // the same network as SCL:
   IF #t1 THEN #f2 := TRUE; END_IF;
END_REGION

REGION Network 10
   Label( azioni )
   RUNG wire#powerrail
      Contact( #f1 )
      S_Coil( #ava )
   END_RUNG
   // the same network as SCL:
   azioni:
   IF #f1 THEN #ava := TRUE; END_IF;
END_REGION

REGION Network 11
   RUNG wire#powerrail
      Contact( #f2 )
      Coil( #ricevuto_ok )
   END_RUNG
   // the same network as SCL:
   #ricevuto_ok := #f2;
END_REGION

REGION Network 12
   RUNG wire#powerrail
      I_Contact( #iniz )
      S_Coil( #iniz )
   END_RUNG
   // the same network as SCL:
   IF NOT #iniz THEN #iniz := TRUE; END_IF;
END_REGION
END_FUNCTION_BLOCK

FUNCTION_BLOCK "Pusher"   // FB5, LAD
{ S7_Optimized_Access := 'TRUE' }
VERSION : 0.1
   VAR_INPUT
      spingi_fine : Bool;
      sens_spingi : Bool;
   END_VAR
   VAR_OUTPUT
      spingi : Bool;
      ferma_nastro : Bool;
      avanti : Bool;
   END_VAR
   VAR
      iniz : Bool;
      f1 : Bool;
      t1 : Bool;
      f2 : Bool;
      t2 : Bool;
      f3 : Bool;
      t3 : Bool;
      sens_spingi_ftrig : F_TRIG;
   END_VAR
BEGIN

REGION Network 1
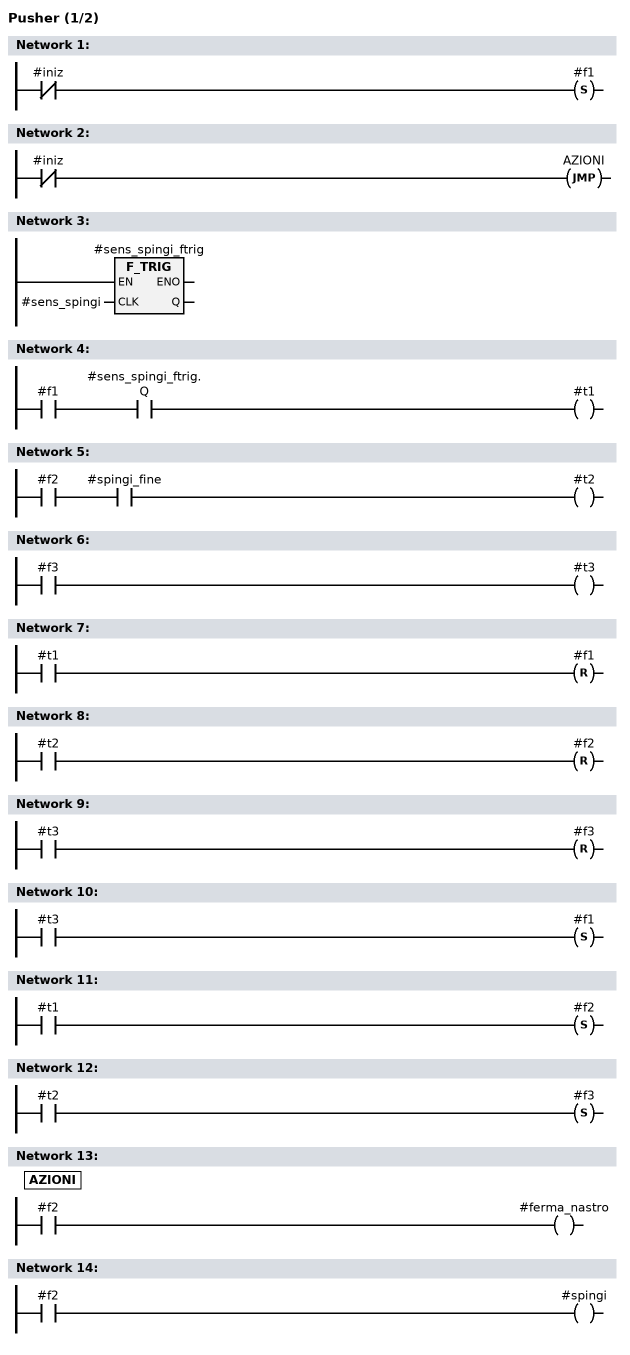
   RUNG wire#powerrail
      I_Contact( #iniz )
      S_Coil( #f1 )
   END_RUNG
   // the same network as SCL:
   IF NOT #iniz THEN #f1 := TRUE; END_IF;
END_REGION

REGION Network 2
   RUNG wire#powerrail
      I_Contact( #iniz )
      JumpCoil( AZIONI )
   END_RUNG
   // the same network as SCL:
   IF NOT #iniz THEN GOTO AZIONI; END_IF;
END_REGION

REGION Network 3
   #sens_spingi_ftrig(CLK := #sens_spingi);   // F_TRIG
END_REGION

REGION Network 4
   RUNG wire#powerrail
      Contact( #f1 )
      Contact( #sens_spingi_ftrig.Q )
      Coil( #t1 )
   END_RUNG
   // the same network as SCL:
   #t1 := #f1 AND #sens_spingi_ftrig.Q;
END_REGION

REGION Network 5
   RUNG wire#powerrail
      Contact( #f2 )
      Contact( #spingi_fine )
      Coil( #t2 )
   END_RUNG
   // the same network as SCL:
   #t2 := #f2 AND #spingi_fine;
END_REGION

REGION Network 6
   RUNG wire#powerrail
      Contact( #f3 )
      Coil( #t3 )
   END_RUNG
   // the same network as SCL:
   #t3 := #f3;
END_REGION

REGION Network 7
   RUNG wire#powerrail
      Contact( #t1 )
      R_Coil( #f1 )
   END_RUNG
   // the same network as SCL:
   IF #t1 THEN #f1 := FALSE; END_IF;
END_REGION

REGION Network 8
   RUNG wire#powerrail
      Contact( #t2 )
      R_Coil( #f2 )
   END_RUNG
   // the same network as SCL:
   IF #t2 THEN #f2 := FALSE; END_IF;
END_REGION

REGION Network 9
   RUNG wire#powerrail
      Contact( #t3 )
      R_Coil( #f3 )
   END_RUNG
   // the same network as SCL:
   IF #t3 THEN #f3 := FALSE; END_IF;
END_REGION

REGION Network 10
   RUNG wire#powerrail
      Contact( #t3 )
      S_Coil( #f1 )
   END_RUNG
   // the same network as SCL:
   IF #t3 THEN #f1 := TRUE; END_IF;
END_REGION

REGION Network 11
   RUNG wire#powerrail
      Contact( #t1 )
      S_Coil( #f2 )
   END_RUNG
   // the same network as SCL:
   IF #t1 THEN #f2 := TRUE; END_IF;
END_REGION

REGION Network 12
   RUNG wire#powerrail
      Contact( #t2 )
      S_Coil( #f3 )
   END_RUNG
   // the same network as SCL:
   IF #t2 THEN #f3 := TRUE; END_IF;
END_REGION

REGION Network 13
   Label( AZIONI )
   RUNG wire#powerrail
      Contact( #f2 )
      Coil( #ferma_nastro )
   END_RUNG
   // the same network as SCL:
   AZIONI:
   #ferma_nastro := #f2;
END_REGION

REGION Network 14
   RUNG wire#powerrail
      Contact( #f2 )
      Coil( #spingi )
   END_RUNG
   // the same network as SCL:
   #spingi := #f2;
END_REGION

REGION Network 15
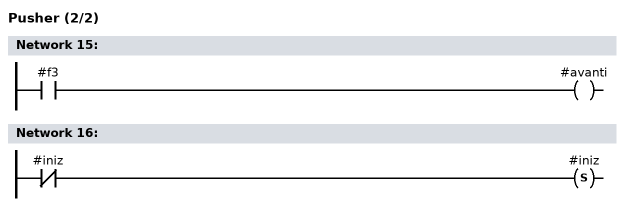
   RUNG wire#powerrail
      Contact( #f3 )
      Coil( #avanti )
   END_RUNG
   // the same network as SCL:
   #avanti := #f3;
END_REGION

REGION Network 16
   RUNG wire#powerrail
      I_Contact( #iniz )
      S_Coil( #iniz )
   END_RUNG
   // the same network as SCL:
   IF NOT #iniz THEN #iniz := TRUE; END_IF;
END_REGION
END_FUNCTION_BLOCK

FUNCTION_BLOCK "Nastro_1"   // FB6, LAD
{ S7_Optimized_Access := 'TRUE' }
VERSION : 0.1
   VAR_INPUT
      ferma : Bool;
      p_dopo : Bool;
      spinto_ok : Bool;
      pronto_consegnare : Bool;
   END_VAR
   VAR_OUTPUT
      push : Bool;
      ava : Bool;
   END_VAR
   VAR
      iniz : Bool;
      f1 : Bool;
      tr1 : Bool;
      F_TRIG_SENS_SPINGI : F_TRIG;
      F_TRIG_PRONTO_CONSEGNARE : F_TRIG;
      tr2 : Bool;
      f2 : Bool;
      tr3 : Bool;
      f3 : Bool;
      tr4 : Bool;
      tr5 : Bool;
      f4 : Bool;
   END_VAR
BEGIN

REGION Network 1
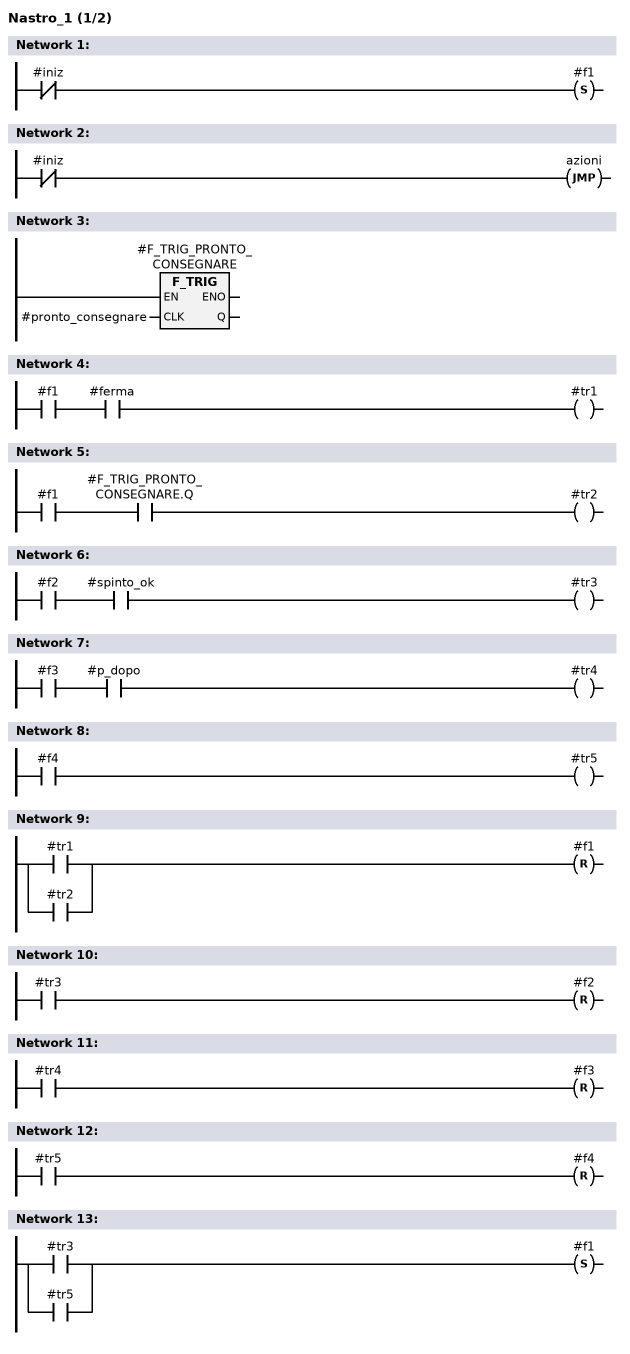
   RUNG wire#powerrail
      I_Contact( #iniz )
      S_Coil( #f1 )
   END_RUNG
   // the same network as SCL:
   IF NOT #iniz THEN #f1 := TRUE; END_IF;
END_REGION

REGION Network 2
   RUNG wire#powerrail
      I_Contact( #iniz )
      JumpCoil( azioni )
   END_RUNG
   // the same network as SCL:
   IF NOT #iniz THEN GOTO azioni; END_IF;
END_REGION

REGION Network 3
   #F_TRIG_PRONTO_CONSEGNARE(CLK := #pronto_consegnare);   // F_TRIG
END_REGION

REGION Network 4
   RUNG wire#powerrail
      Contact( #f1 )
      Contact( #ferma )
      Coil( #tr1 )
   END_RUNG
   // the same network as SCL:
   #tr1 := #f1 AND #ferma;
END_REGION

REGION Network 5
   RUNG wire#powerrail
      Contact( #f1 )
      Contact( #F_TRIG_PRONTO_CONSEGNARE.Q )
      Coil( #tr2 )
   END_RUNG
   // the same network as SCL:
   #tr2 := #f1 AND #F_TRIG_PRONTO_CONSEGNARE.Q;
END_REGION

REGION Network 6
   RUNG wire#powerrail
      Contact( #f2 )
      Contact( #spinto_ok )
      Coil( #tr3 )
   END_RUNG
   // the same network as SCL:
   #tr3 := #f2 AND #spinto_ok;
END_REGION

REGION Network 7
   RUNG wire#powerrail
      Contact( #f3 )
      Contact( #p_dopo )
      Coil( #tr4 )
   END_RUNG
   // the same network as SCL:
   #tr4 := #f3 AND #p_dopo;
END_REGION

REGION Network 8
   RUNG wire#powerrail
      Contact( #f4 )
      Coil( #tr5 )
   END_RUNG
   // the same network as SCL:
   #tr5 := #f4;
END_REGION

REGION Network 9
   RUNG wire#powerrail
      Contact( #tr1 )
      wire#w1
      R_Coil( #f1 )
   END_RUNG
   RUNG wire#powerrail
      Contact( #tr2 )
   END_RUNG wire#w1
   // the same network as SCL:
   IF #tr1 OR #tr2 THEN #f1 := FALSE; END_IF;
END_REGION

REGION Network 10
   RUNG wire#powerrail
      Contact( #tr3 )
      R_Coil( #f2 )
   END_RUNG
   // the same network as SCL:
   IF #tr3 THEN #f2 := FALSE; END_IF;
END_REGION

REGION Network 11
   RUNG wire#powerrail
      Contact( #tr4 )
      R_Coil( #f3 )
   END_RUNG
   // the same network as SCL:
   IF #tr4 THEN #f3 := FALSE; END_IF;
END_REGION

REGION Network 12
   RUNG wire#powerrail
      Contact( #tr5 )
      R_Coil( #f4 )
   END_RUNG
   // the same network as SCL:
   IF #tr5 THEN #f4 := FALSE; END_IF;
END_REGION

REGION Network 13
   RUNG wire#powerrail
      Contact( #tr3 )
      wire#w1
      S_Coil( #f1 )
   END_RUNG
   RUNG wire#powerrail
      Contact( #tr5 )
   END_RUNG wire#w1
   // the same network as SCL:
   IF #tr3 OR #tr5 THEN #f1 := TRUE; END_IF;
END_REGION

REGION Network 14
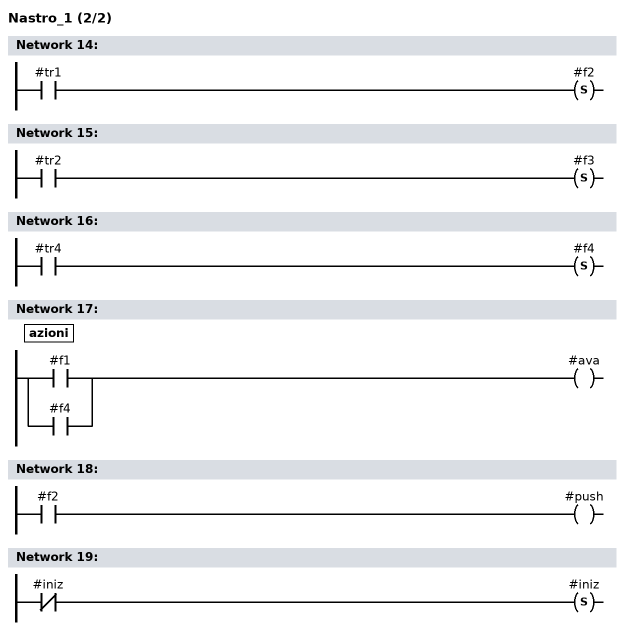
   RUNG wire#powerrail
      Contact( #tr1 )
      S_Coil( #f2 )
   END_RUNG
   // the same network as SCL:
   IF #tr1 THEN #f2 := TRUE; END_IF;
END_REGION

REGION Network 15
   RUNG wire#powerrail
      Contact( #tr2 )
      S_Coil( #f3 )
   END_RUNG
   // the same network as SCL:
   IF #tr2 THEN #f3 := TRUE; END_IF;
END_REGION

REGION Network 16
   RUNG wire#powerrail
      Contact( #tr4 )
      S_Coil( #f4 )
   END_RUNG
   // the same network as SCL:
   IF #tr4 THEN #f4 := TRUE; END_IF;
END_REGION

REGION Network 17
   Label( azioni )
   RUNG wire#powerrail
      Contact( #f1 )
      wire#w1
      Coil( #ava )
   END_RUNG
   RUNG wire#powerrail
      Contact( #f4 )
   END_RUNG wire#w1
   // the same network as SCL:
   azioni:
   #ava := #f1 OR #f4;
END_REGION

REGION Network 18
   RUNG wire#powerrail
      Contact( #f2 )
      Coil( #push )
   END_RUNG
   // the same network as SCL:
   #push := #f2;
END_REGION

REGION Network 19
   RUNG wire#powerrail
      I_Contact( #iniz )
      S_Coil( #iniz )
   END_RUNG
   // the same network as SCL:
   IF NOT #iniz THEN #iniz := TRUE; END_IF;
END_REGION
END_FUNCTION_BLOCK

FUNCTION "MHJ-PLC-Lab-Function-S71200" : Void   // FC9000, SCL
{ S7_Optimized_Access := 'TRUE' }
VERSION : 0.1
   VAR_TEMP
      rdTimeReturn : Int;
      outputTime : DTL;
      SyncVal : Byte;
      forVal : Int;
      forVal_2 : Int;
      Value : Byte;
   END_VAR
   VAR CONSTANT
      CompVal : Byte := 16#34;
      Value_01 : Byte := 16#11;
      Value_01_DW : DWord := 16#A165_D992;
      Value_02_DW : DWord := 16#58BE_4401;
   END_VAR
BEGIN

   #Value:=PEEK(area := 16#82,
        dbNumber := 0,
        byteOffset := 511);
   #Value := #Value + 1;

   POKE(area := 16#82,
        dbNumber := 0,
        byteOffset := 511,
        value := #Value);

   POKE(area:=16#81,
        dbNumber:=0,
        byteOffset:=1016,
        value:=#Value_01_DW);
   POKE(area := 16#81,
        dbNumber := 0,
        byteOffset := 1020,
        value := #Value_02_DW);

   POKE(area := 16#81,
        dbNumber := 0,
        byteOffset := 511,
        value := B#16#00);

   FOR #forVal := 0 TO 120 DO
       FOR #forVal_2:=0 TO 10 DO
           #rdTimeReturn:=RD_SYS_T(#outputTime);
           #rdTimeReturn := WR_SYS_T(#outputTime);
           #rdTimeReturn := RD_SYS_T(#outputTime);
           #rdTimeReturn := WR_SYS_T(#outputTime);
       END_FOR;
       #SyncVal:= PEEK(area := 16#81,
                      dbNumber := 0,
                      byteOffset := 511);
       IF #SyncVal = #CompVal THEN
          GOTO M_1;
       END_IF;
   END_FOR;
   RETURN;

   M_1:
   POKE(area := 16#81,
        dbNumber := 0,
        byteOffset := 511,
        value := B#16#0);
END_FUNCTION

ORGANIZATION_BLOCK "Main"   // OB1, LAD, ProgramCycle
TITLE = "Main Program Sweep (Cycle)"
{ S7_Optimized_Access := 'TRUE' }
VERSION : 0.1
   VAR_INPUT
      Initial_Call : Bool;   // Initial call of this OB
      Remanence : Bool;   // =True, if remanent data are available
   END_VAR
   VAR_TEMP   // added for the SCL form of the ladder/FBD networks
      _w1 : Bool;
   END_VAR
BEGIN

REGION Network 1: Konnektierungsbaustein für PLC-Lab
   // Im Netzwerk 1 wird der Konnektierungsbaustein für PLC-Lab aufgerufen.
   // Dieser Aufruf darf nicht entfernt werden!
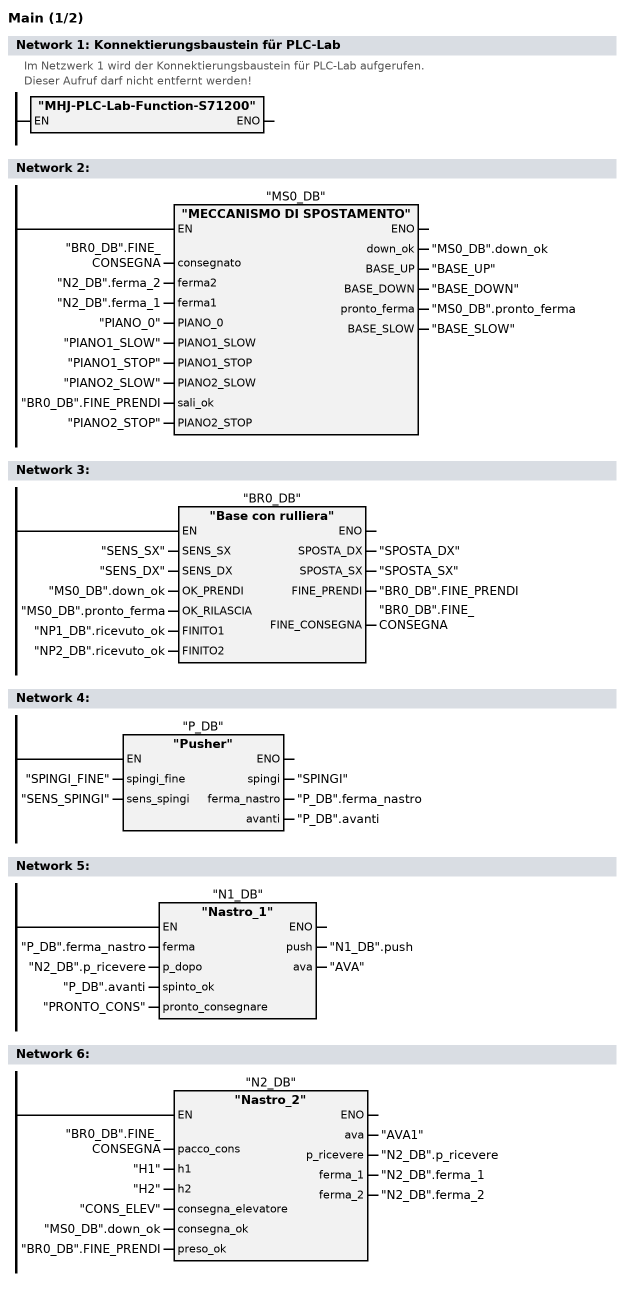
   RUNG wire#powerrail
      "MHJ-PLC-Lab-Function-S71200"()
   END_RUNG
   // the same network as SCL:
   "MHJ-PLC-Lab-Function-S71200"();
END_REGION

REGION Network 2
   RUNG wire#powerrail
      "MS0_DB"(consegnato := "BR0_DB".FINE_CONSEGNA, ferma2 := "N2_DB".ferma_2, ferma1 := "N2_DB".ferma_1, PIANO_0 := "PIANO_0", PIANO1_SLOW := "PIANO1_SLOW", PIANO1_STOP := "PIANO1_STOP", PIANO2_SLOW := "PIANO2_SLOW", sali_ok := "BR0_DB".FINE_PRENDI, PIANO2_STOP := "PIANO2_STOP", down_ok => "MS0_DB".down_ok, BASE_UP => "BASE_UP", BASE_DOWN => "BASE_DOWN", pronto_ferma => "MS0_DB".pronto_ferma, BASE_SLOW => "BASE_SLOW")
   END_RUNG
   // the same network as SCL:
   "MS0_DB"(consegnato := "BR0_DB".FINE_CONSEGNA,   // "MECCANISMO DI SPOSTAMENTO"
            ferma2 := "N2_DB".ferma_2,
            ferma1 := "N2_DB".ferma_1,
            PIANO_0 := "PIANO_0",
            PIANO1_SLOW := "PIANO1_SLOW",
            PIANO1_STOP := "PIANO1_STOP",
            PIANO2_SLOW := "PIANO2_SLOW",
            sali_ok := "BR0_DB".FINE_PRENDI,
            PIANO2_STOP := "PIANO2_STOP",
            down_ok => "MS0_DB".down_ok,
            BASE_UP => "BASE_UP",
            BASE_DOWN => "BASE_DOWN",
            pronto_ferma => "MS0_DB".pronto_ferma,
            BASE_SLOW => "BASE_SLOW");
END_REGION

REGION Network 3
   RUNG wire#powerrail
      "BR0_DB"(SENS_SX := "SENS_SX", SENS_DX := "SENS_DX", OK_PRENDI := "MS0_DB".down_ok, OK_RILASCIA := "MS0_DB".pronto_ferma, FINITO1 := "NP1_DB".ricevuto_ok, FINITO2 := "NP2_DB".ricevuto_ok, SPOSTA_DX => "SPOSTA_DX", SPOSTA_SX => "SPOSTA_SX", FINE_PRENDI => "BR0_DB".FINE_PRENDI, FINE_CONSEGNA => "BR0_DB".FINE_CONSEGNA)
   END_RUNG
   // the same network as SCL:
   "BR0_DB"(SENS_SX := "SENS_SX",   // "Base con rulliera"
            SENS_DX := "SENS_DX",
            OK_PRENDI := "MS0_DB".down_ok,
            OK_RILASCIA := "MS0_DB".pronto_ferma,
            FINITO1 := "NP1_DB".ricevuto_ok,
            FINITO2 := "NP2_DB".ricevuto_ok,
            SPOSTA_DX => "SPOSTA_DX",
            SPOSTA_SX => "SPOSTA_SX",
            FINE_PRENDI => "BR0_DB".FINE_PRENDI,
            FINE_CONSEGNA => "BR0_DB".FINE_CONSEGNA);
END_REGION

REGION Network 4
   RUNG wire#powerrail
      "P_DB"(spingi_fine := "SPINGI_FINE", sens_spingi := "SENS_SPINGI", spingi => "SPINGI", ferma_nastro => "P_DB".ferma_nastro, avanti => "P_DB".avanti)
   END_RUNG
   // the same network as SCL:
   "P_DB"(spingi_fine := "SPINGI_FINE",   // "Pusher"
          sens_spingi := "SENS_SPINGI",
          spingi => "SPINGI",
          ferma_nastro => "P_DB".ferma_nastro,
          avanti => "P_DB".avanti);
END_REGION

REGION Network 5
   RUNG wire#powerrail
      "N1_DB"(ferma := "P_DB".ferma_nastro, p_dopo := "N2_DB".p_ricevere, spinto_ok := "P_DB".avanti, pronto_consegnare := "PRONTO_CONS", push => "N1_DB".push, ava => "AVA")
   END_RUNG
   // the same network as SCL:
   "N1_DB"(ferma := "P_DB".ferma_nastro,   // "Nastro_1"
           p_dopo := "N2_DB".p_ricevere,
           spinto_ok := "P_DB".avanti,
           pronto_consegnare := "PRONTO_CONS",
           push => "N1_DB".push,
           ava => "AVA");
END_REGION

REGION Network 6
   RUNG wire#powerrail
      "N2_DB"(pacco_cons := "BR0_DB".FINE_CONSEGNA, h1 := "H1", h2 := "H2", consegna_elevatore := "CONS_ELEV", consegna_ok := "MS0_DB".down_ok, preso_ok := "BR0_DB".FINE_PRENDI, ava => "AVA1", p_ricevere => "N2_DB".p_ricevere, ferma_1 => "N2_DB".ferma_1, ferma_2 => "N2_DB".ferma_2)
   END_RUNG
   // the same network as SCL:
   "N2_DB"(pacco_cons := "BR0_DB".FINE_CONSEGNA,   // "Nastro_2"
           h1 := "H1",
           h2 := "H2",
           consegna_elevatore := "CONS_ELEV",
           consegna_ok := "MS0_DB".down_ok,
           preso_ok := "BR0_DB".FINE_PRENDI,
           ava => "AVA1",
           p_ricevere => "N2_DB".p_ricevere,
           ferma_1 => "N2_DB".ferma_1,
           ferma_2 => "N2_DB".ferma_2);
END_REGION

REGION Network 7
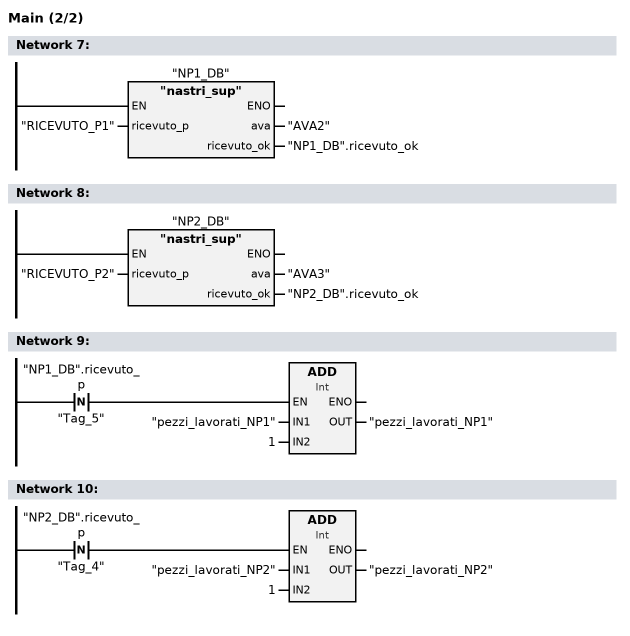
   RUNG wire#powerrail
      "NP1_DB"(ricevuto_p := "RICEVUTO_P1", ava => "AVA2", ricevuto_ok => "NP1_DB".ricevuto_ok)
   END_RUNG
   // the same network as SCL:
   "NP1_DB"(ricevuto_p := "RICEVUTO_P1", ava => "AVA2", ricevuto_ok => "NP1_DB".ricevuto_ok);   // "nastri_sup"
END_REGION

REGION Network 8
   RUNG wire#powerrail
      "NP2_DB"(ricevuto_p := "RICEVUTO_P2", ava => "AVA3", ricevuto_ok => "NP2_DB".ricevuto_ok)
   END_RUNG
   // the same network as SCL:
   "NP2_DB"(ricevuto_p := "RICEVUTO_P2", ava => "AVA3", ricevuto_ok => "NP2_DB".ricevuto_ok);   // "nastri_sup"
END_REGION

REGION Network 9
   RUNG wire#powerrail
      N_Contact(operand := "NP1_DB".ricevuto_p, bit := "Tag_5")
      { S7_Templates := "SrcType := Int" } Add(in1 := "pezzi_lavorati_NP1", in2 := 1, out => "pezzi_lavorati_NP1")
   END_RUNG
   // the same network as SCL:
   #_w1 := NOT "NP1_DB".ricevuto_p AND "Tag_5";   // falling edge of "NP1_DB".ricevuto_p
   "Tag_5" := "NP1_DB".ricevuto_p;
   IF #_w1 THEN "pezzi_lavorati_NP1" := "pezzi_lavorati_NP1" + 1; END_IF;
END_REGION

REGION Network 10
   RUNG wire#powerrail
      N_Contact(operand := "NP2_DB".ricevuto_p, bit := "Tag_4")
      { S7_Templates := "SrcType := Int" } Add(in1 := "pezzi_lavorati_NP2", in2 := 1, out => "pezzi_lavorati_NP2")
   END_RUNG
   // the same network as SCL:
   #_w1 := NOT "NP2_DB".ricevuto_p AND "Tag_4";   // falling edge of "NP2_DB".ricevuto_p
   "Tag_4" := "NP2_DB".ricevuto_p;
   IF #_w1 THEN "pezzi_lavorati_NP2" := "pezzi_lavorati_NP2" + 1; END_IF;
END_REGION
END_ORGANIZATION_BLOCK

(* ===== HMI "HMI_RT_1" =====
system functions are stored by id; their names below are inferred from use
connection "HMI_Connection_1": ETHERNET, S7_1200_OMS

HMI tags "Default tag table"
   "Tag_ScreenNumber" : UInt, internal
   "PIANO_0" : Bool = PLC PIANO_0 AT %I0.2, 1 s
   "N2_DB_p_ricevere" : Bool = PLC N2_DB.p_ricevere, 1 s
   "N1_DB_ava" : Bool = PLC N1_DB.ava, 1 s
   "P_DB_spingi" : Bool = PLC P_DB.spingi, 1 s
   "pezzi_lavorati_NP1" : Int = PLC pezzi_lavorati_NP1 AT %MW16, 1 s
   "pezzi_lavorati_NP2" : Int = PLC pezzi_lavorati_NP2 AT %MW18, 1 s

screen "Root screen" 800x420, template "Template_1"
   on GenerateScreen: SetTag("Tag_ScreenNumber", 1)
   TextField "Text field_1" at 0,19 size 672x29; Text 'PIANO 1 , PACCHI CONSEGNATI:'
   TextField "Text field_2" at 0,51 size 609x29; Text 'PIANO 2 , PACCHI CONSEGNATI:'
   Circle "Circle_1" at 750,151 size 31x31
      Appearance <- "PIANO_0"
   TextField "Text field_3" at 511,84 size 222x154; Text 'STATO ELEVATORE'
   TextField "Text field_4" at 39,92 size 173x29; Text 'PIANO 0:'
   TextField "Text field_5" at 35,127 size 291x29; Text 'STATO NASTRO 2'
   TextField "Text field_6" at 35,189 size 291x29; Text 'STATO NASTRO 1'
   TextField "Text field_7" at 38,260 size 293x32; Text 'STATO PUSHER'
   IOField "I/O field_1" at 699,16 size 96x32; FormatPattern 999
      ProcessValue <- "pezzi_lavorati_NP1"
   IOField "I/O field_2" at 699,48 size 96x32; FormatPattern 999
      ProcessValue <- "pezzi_lavorati_NP2"
   Circle "Circle_2" at 359,126 size 31x31
      Appearance <- "N2_DB_p_ricevere"
   Circle "Circle_3" at 359,187 size 31x31
      Appearance <- "N1_DB_ava"
   Circle "Circle_4" at 360,260 size 31x31
      Appearance <- "P_DB_spingi"

Template "Template_1" 800x420
   Button "Exit" at 720,360 size 78x58; TextOff 'Exit'; PictureOff "ExitRuntime_TP900_Comfort_TR"; PictureOn "ExitRuntime_TP900_Comfort_TR"
      on Release: StopRuntime(0)
   Button "Template_Button" at 640,360 size 78x58; TextOff 'Text'
   Button "Template_Button_1" at 560,360 size 78x58; TextOff 'Text'
   Button "Template_Button_2" at 480,360 size 78x58; TextOff 'Text'
   Button "Template_Button_3" at 400,360 size 78x58; TextOff 'Text'
   Button "Template_Button_4" at 321,360 size 78x58; TextOff 'Text'
   Button "Template_Button_5" at 241,360 size 78x58; TextOff 'Text'
   Button "Template_Button_6" at 161,360 size 78x58; TextOff 'Text'
   Button "Alarms" at 81,360 size 78x58; TextOff 'Alarms'; PictureOff "AlarmDisplay_TP900_Comfort_TR"; PictureOn "AlarmDisplay_TP900_Comfort_TR"
      on Release: function_ef3f5d25("Alarm window_Unacknowledged", -1)
   Button "Start screen" at 1,360 size 78x58; TextOff 'Start screen'; PictureOff "NavigateHome_TP900_Comfort_TR"; PictureOn "NavigateHome_TP900_Comfort_TR"
      on Release: ActivateScreen("Root screen", 0)
*)